DEVICE_TYPE _WaterHeater
  (* Standard: 61499-2 *)
  (* Version 0.1, 2017-00-25, hpea485, UOA *)
  RESOURCE controller : _WaterHeaterController
  END_RESOURCE
  RESOURCE plant : _WaterHeaterPlant
  END_RESOURCE
END_DEVICE_TYPE
